// TwinCAT 3 PLC project Hola_Mundo_PLC
// ProgramVersion: 3.1.4024.0
// libraries:
//   Tc2_Standard, * (Beckhoff Automation GmbH)
//   Tc2_System, * (Beckhoff Automation GmbH)
//   Tc3_Module, * (Beckhoff Automation GmbH)
//   VisuDialogs, * (System)
// project tree:
//   / GlobalTextList.TcGTLO, PlcTask.TcTTO, Visualization Manager.TcVMO (not stored)
//   POUs/ MAIN.TcPOU
//   VISUs/ V_Hola_Mundo.TcVIS
// real-time tasks:
//   TASK PlcTask: cycle T#10ms, priority 20, ADS port 350
// I/O:
//   DEVICE Device 1 (EtherCAT) (disabled), AmsNetId 5.132.11.217.2.1
//     Term 1 (EK1200) [EK1200-5000 EtherCAT Power supply (2A E-Bus)]
//       Term 2 (EL1008) [EL1008 8Ch. Dig. Input 24V, 3ms]
//       Term 3 (EL2004) [EL2004 4Ch. Dig. Output 24V, 0.5A]
//       Term 4 (EL9011) [EL9011 End Terminal]
// variable links:
//   Hola_Mundo_PLC/Hola_Mundo_PLC Instance <-> Device 1 (EtherCAT)/Term 1 (EK1200)/Term 2 (EL1008)
//     PlcTask Inputs/MAIN.i_Pulsador <-> Channel 1/Pulsador
//   Hola_Mundo_PLC/Hola_Mundo_PLC Instance <-> Device 1 (EtherCAT)/Term 1 (EK1200)/Term 3 (EL2004)
//     PlcTask Outputs/MAIN.o_Lampara <-> Channel 1/Lampara

CONFIGURATION Hola_Mundo_PLC
    RESOURCE PLC ON TwinCAT3
        TASK PlcTask(INTERVAL := T#10ms, PRIORITY := 20);
        PROGRAM MAIN WITH PlcTask : MAIN;
    END_RESOURCE
END_CONFIGURATION

// ---- POUs/MAIN.TcPOU
// Hola Mundo de la Programación de PLC
PROGRAM MAIN
VAR
    ContadorCiclos: UINT;
    i_Pulsador AT %I* : BOOL;
    o_Lampara  AT %Q* : BOOL;
    
END_VAR

ContadorCiclos := ContadorCiclos + 1;
o_Lampara := i_Pulsador;

END_PROGRAM

// ---- GlobalTextList.TcGTLO
TEXTLIST GlobalTextList
  139 = '%d'
  179 = 'Contador'
  944 = 'DEMO'
  553 = 'HOLA MUNDO'
  116 = 'Lámpara'
  279 = 'Pulsador'
  466 = 'Reinicia'
END_TEXTLIST

// ---- VISUs/V_Hola_Mundo.TcVIS
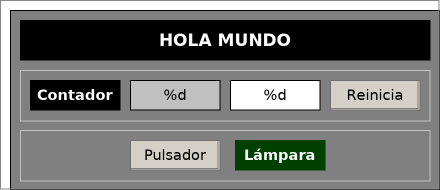
VISUALIZATION V_Hola_Mundo  // 440x190
    Rectangle (10,10 430x180)
    Rectangle (20,70 410x51)
    Rectangle (20,130 410x51)
    Rectangle (20,20 410x40), "HOLA MUNDO"
    Rectangle (30,80 90x30), "Contador"
    Rectangle (230,80 90x30), "%d", text variable: MAIN.ContadorCiclos
        OnMouseClick: write the text variable via Default
    Rectangle (130,80 90x30), "%d", text variable: MAIN.ContadorCiclos
    Button (330,80 90x30), "Reinicia"
        OnMouseClick: execute { MAIN.ContadorCiclos := 0; }
    Button (130,140 90x30), "Pulsador"
        tap MAIN.i_Pulsador
    Rectangle (235,140 90x30), "Lámpara", colour toggle: MAIN.o_Lampara
END_VISUALIZATION
